PROGRAM prgCom
VAR
	fbCom		: FB_MqttCommunicator;
END_VAR

fbCom(
	bConnect:= TRUE, 
	sUserName:= 'f9df9331-ad26-4233-a90b-1145ad47a6fc', 
	sUserPassword:= '508d778d-b673-4a9a-b271-2192eb65a63c', 
	eSavePositionCertificate:= eSavePositionOnPLC.ePostionC, 
	bConnected=> , 
	bError=> , 
	hrErrorCode=> , 
	eConnectionState=> , 
	eErrorMessage_Out=> );

END_PROGRAM

(* stored: Version 1.1.0.1, ProductVersion 3.1.4024.9
   POU prgCom: Id {59faba11-cfd9-4afc-bef7-e44e928da019}, SpecialFunc None *)
